(* PLC project prj, KAIST_DSLAB noNameNow 1, author bwkim *)
(* stored: creationDateTime 2015-9-4T03:02:16, modificationDateTime 2015-9-4T03:02:16 *)

PROGRAM Program1____R_TRIG_and_SR
  VAR
    R_TRIG_Switch : null;
  END_VAR
  VAR
    SR_Manu : null;
  END_VAR
  VAR
    SR_Manual : null;
  END_VAR
  VAR_IN_OUT
    cmdManual : BOOL := FALSE;
  END_VAR

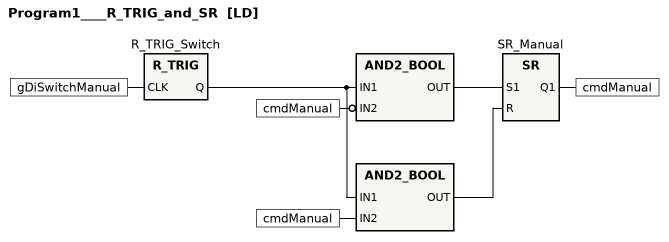
(* LD diagram, written out as Structured Text *)
R_TRIG_Switch(CLK := gDiSwitchManual);
SR_Manual(S1 := AND2_BOOL(R_TRIG_Switch.Q, NOT cmdManual), R := AND2_BOOL(R_TRIG_Switch.Q, cmdManual));
cmdManual := SR_Manual.Q1;
END_PROGRAM
